// TIA Portal V17 export
// export: Created 2023-02-13T11:16:05.3142725Z, ExportSetting WithDefaults, DisplayName Totally Integrated Automation Portal, DisplayVersion V17, DisplayName TIA Portal Openness, DisplayVersion V17, DisplayName TIA Portal Teamcenter Gateway, DisplayVersion V17, DisplayName TIA Portal Version Control Interface, DisplayVersion V17, DisplayName SINAMICS Startdrive Advanced, DisplayVersion V17, DisplayName SINAMICS Startdrive G130, G150, S120, S150, SINAMICS MV, S210, DisplayVersion V17, DisplayName SINAMICS Startdrive G110M, G120, G120C, G120D, G120P, G115D, DisplayVersion V17, DisplayName STEP 7 Professional, DisplayVersion V17, DisplayName STEP 7 Safety, DisplayVersion V17, DisplayName WinCC Professional, DisplayVersion V17
DATA_BLOCK "Sugar to Mix"   // DB231
{ S7_Optimized_Access := 'FALSE' }
VERSION : 0.1
// stored: AutoNumber false, DBAccessibleFromOPCUA true, DBAccessibleFromWebserver true, IsOnlyStoredInLoadMemory false, IsWriteProtectedInAS false
   VAR
      HeartBeat : Bool;   // Alternating value of 0 and 1 to indicate that the PLC is alive
      "System ready to run" : Bool;   // Scala system is ready to receive signal from customer
      "Transfer in process" : Bool;   // transfer in process
      "Transfer completed" : Bool;   // transfer completed
      "Transfer alarm" : Bool;   // warning alarm exist (Conveying timeout, Filling timeout, etc)
      "Weight Actual for Mixer" : Real;
   END_VAR
BEGIN
END_DATA_BLOCK
